// TIA Portal project "Onlab" (V16)

(* hardware
DEVICE "S71500/ET200MP station_1"  S7-1500 station
   slot 0: "Rail_0"  Rack  6ES7 590-1***0-0AA0
   slot 1: "PLC_1"  CPU 1515-2 PN  6ES7 515-2AM00-0AB0  V1.8
      slot 3: "CPU display_1"  6ES7591-1BA00-0AA0
      slot 32768: "PROFINET interface_1"  X1
         slot 32769: "Port_1"  X1 P1
         slot 32770: "Port_2"  X1 P2
      slot 33024: "PROFINET interface_2"  X2
         slot 33025: "Port_1"  X2 P1
*)

// ===== PLC "PLC_1"  CPU 1515-2 PN =====

VAR_GLOBAL   // PLC tag table "Default tag table"
   "Start" AT %I0.0 : Bool;
   "ST10_SMD" AT %I0.1 : Bool;
   "ST10_SED" AT %I0.2 : Bool;
   "ST10_SRD" AT %I0.3 : Bool;
   "ST20_SMD" AT %I0.4 : Bool;
   "ST20_SRD" AT %I0.5 : Bool;
   "ST20_SED" AT %I0.6 : Bool;
   "ST30_SMD" AT %I0.7 : Bool;
   "ST30_SRD" AT %I1.0 : Bool;
   "ST30_SED" AT %I1.1 : Bool;
   "Start2" AT %I1.2 : Bool;
END_VAR

DATA_BLOCK "PLC_PRG_DB"   // DB1
{ S7_Optimized_Access := 'TRUE' }
VERSION : 0.1
   VAR
      startp : Bool;
      start2p : Bool;
      st10smdp : Bool;
      st10srdp : Bool;
      st10sedp : Bool;
      st20smdp : Bool;
      st20srdp : Bool;
      st20sedp : Bool;
      st30smdp : Bool;
      st30srdp : Bool;
      st30sedp : Bool;
      st40smdp : Bool;
      st40srdp : Bool;
      st40sedp : Bool;
      st20recrdy : Bool;
      st30recrdy : Bool;
      st40recrdy : Bool;
   END_VAR
BEGIN
END_DATA_BLOCK

DATA_BLOCK "ST10"   // DB9
{ S7_Optimized_Access := 'TRUE' }
VERSION : 0.1
// stored: InstanceOfName CB
"CB"
BEGIN
END_DATA_BLOCK

DATA_BLOCK "ST20"   // DB10
{ S7_Optimized_Access := 'TRUE' }
VERSION : 0.1
// stored: InstanceOfName CB
"CB"
BEGIN
END_DATA_BLOCK

DATA_BLOCK "ST30"   // DB11
{ S7_Optimized_Access := 'TRUE' }
VERSION : 0.1
// stored: InstanceOfName CB
"CB"
BEGIN
END_DATA_BLOCK

DATA_BLOCK "ST40_db"   // DB12
{ S7_Optimized_Access := 'TRUE' }
VERSION : 0.1
// stored: InstanceOfName CB
"CB"
BEGIN
END_DATA_BLOCK

DATA_BLOCK "ST50"   // DB13
{ S7_Optimized_Access := 'TRUE' }
VERSION : 0.1
// stored: InstanceOfName CB
"CB"
BEGIN
END_DATA_BLOCK

DATA_BLOCK "ST60"   // DB14
{ S7_Optimized_Access := 'TRUE' }
VERSION : 0.1
// stored: InstanceOfName CB
"CB"
BEGIN
END_DATA_BLOCK

DATA_BLOCK "ST70"   // DB15
{ S7_Optimized_Access := 'TRUE' }
VERSION : 0.1
// stored: InstanceOfName CB
"CB"
BEGIN
END_DATA_BLOCK

// folder: DBk

DATA_BLOCK "ST10_DBaaa"   // DB2
{ S7_Optimized_Access := 'TRUE' }
VERSION : 0.1
   VAR
      Szenzor1 : Bool;   // Optikai szenzor új darab érz. (bemenet)
      Szenzor2 : Bool;   // Lassító szenzor (bemenet)
      Szenzor3 : Bool;   // Megállító szenzor (bemenet)
      NyG : Bool;   // Nyomógomb a pálya elindításához (bemenet)
      Fényv : Bool;   // Fény visszajelzés az operátornak (kimenet)
      Motor100 : Bool;   // Motor 100% sebességgel (kimenet)
      Motor50 : Bool;   // Motor 50% sebességgel (kimenet)
      MotorStop : Bool;   // Motor áll (kimenet)
      NyGPOSEDGE : Bool;   // NyG felfutóél boolja (belső változó)
      Rdy : Bool;   // ST10 Kész új darab fogadására (kimenet)
      Vonalkód : Struct   // Termelésirányításnak átadott adat (kimenet)
         kód : Array[0..7] of Char;
         feldolgozva : Bool;
      END_STRUCT;
      "Kapott adat" : Struct   // Termelésirányítástól kapott információk (bemenet)
         kód : Array[0..7] of Char;
         "új darab" : Bool;
         Levegő : Bool;
         Fény : Bool;
         Visszajáratott : Bool;
      END_STRUCT;
      Állapotok : Array[0..4] of Bool;   // Az állomás állapotai (belső változó)
   END_VAR
BEGIN
   // Állapotok[0] : Várás
   // Állapotok[1] : Motor100
   // Állapotok[2] : Motor50
   // Állapotok[3] : MotorStop
   // Állapotok[4] : Kiadás
END_DATA_BLOCK

DATA_BLOCK "ST20_DBaaa"   // DB3
{ S7_Optimized_Access := 'TRUE' }
VERSION : 0.1
   VAR
      Szenzor1 : Bool := false;   // Lassító szenzor (bemenet)
      Szenzor2 : Bool := false;   // Megállító szenzor (bemenet)
      Vízsz : Bool := false;   // Végállás érz. (bemenet)
      Függ : Bool := false;   // Végállás érz. (bemenet)
      Motor100 : Bool := false;   // Motor 100% sebességgel (kimenet)
      Motor50 : Bool := false;   // Motor 50% sebességgel (kimenet)
      MotorStop : Bool := false;   // Motor áll (kimenet)
      NyGPOSEDGE : Bool := false;   // NyG felfutóél boolja (belső változó)
      Rdy : Bool;   // ST20 Kész új darab fogadására (kimenet)
      Vonalkód : Struct   // Termelésirányításnak átadott adat (kimenet)
         kód : Array[0..7] of Char;
         feldolgozva : Bool;
      END_STRUCT;
      "Kapott adat" : Struct   // Termelésirányítástól kapott információk (bemenet)
         kód : Array[0..7] of Char;
         "új darab" : Bool;
         Levegő : Bool;
         Fény : Bool;
         Visszajáratott : Bool;
      END_STRUCT;
      Állapotok : Array[0..5] of Bool;   // Az állomás állapotai (belső változó)
   END_VAR
BEGIN
   // Állapotok[0] : Várás
   // Állapotok[1] : Motor100
   // Állapotok[2] : Motor50
   // Állapotok[3] : MotorStop
   // Állapotok[4] : ST30 felé
   // Állapotok[5] : ST60 felé
END_DATA_BLOCK

DATA_BLOCK "ST30_DBaaa"   // DB4
{ S7_Optimized_Access := 'TRUE' }
VERSION : 0.1
   VAR
      Szenzor1 : Bool := false;   // Lassító szenzor (bemenet)
      Szenzor2 : Bool := false;   // Megállító szenzor (bemenet)
      Vízsz : Bool := false;   // Végállás érz. (bemenet)
      Függ : Bool := false;   // Végállás érz. (bemenet)
      Motor100 : Bool := false;   // Motor 100% sebességgel (kimenet)
      Motor50 : Bool := false;   // Motor 50% sebességgel (kimenet)
      MotorStop : Bool := false;   // Motor áll (kimenet)
      NyGPOSEDGE : Bool := false;   // NyG felfutóél boolja (belső változó)
      Rdy : Bool;   // ST30 Kész új darab fogadására (kimenet)
      Vonalkód : Struct   // Termelésirányításnak átadott adat (kimenet)
         kód : Array[0..7] of Char;
         feldolgozva : Bool;
      END_STRUCT;
      "Kapott adat" : Struct   // Termelésirányítástól kapott információk (bemenet)
         kód : Array[0..7] of Char;
         "új darab" : Bool;
         Levegő : Bool;
         Fény : Bool;
         Visszajáratott : Bool;
      END_STRUCT;
      Állapotok : Array[0..5] of Bool;   // Az állomás állapotai (belső változó)
   END_VAR
BEGIN
   // Állapotok[0] : Várás
   // Állapotok[1] : Motor100
   // Állapotok[2] : Motor50
   // Állapotok[3] : MotorStop
   // Állapotok[4] : ST30 felé
   // Állapotok[5] : ST60 felé
END_DATA_BLOCK

DATA_BLOCK "ST40_DBaaa"   // DB5
{ S7_Optimized_Access := 'TRUE' }
VERSION : 0.1
   VAR
      Szenzor1 : Bool := false;   // Lassító szenzor (bemenet)
      Szenzor2 : Bool := false;   // Megállító szenzor (bemenet)
      Felső : Bool := false;   // Végállás érz. (bemenet)
      Alsó : Bool := false;   // Végállás érz. (bemenet)
      Motor100 : Bool := false;   // Motor 100% sebességgel (kimenet)
      Motor50 : Bool := false;   // Motor 50% sebességgel (kimenet)
      MotorStop : Bool := false;   // Motor áll (kimenet)
      NyGPOSEDGE : Bool := false;   // NyG felfutóél boolja (belső változó)
      Rdy : Bool;   // ST40 Kész új darab fogadására (kimenet)
      KiadásRdy : Bool;
      Vonalkód : Struct   // Termelésirányításnak átadott adat (kimenet)
         kód : Array[0..7] of Char;
         feldolgozva : Bool;
      END_STRUCT;
      "Kapott adat" : Struct   // Termelésirányítástól kapott információk (bemenet)
         kód : Array[0..7] of Char;
         "új darab" : Bool;
         Levegő : Bool;
         Fény : Bool;
         Visszajáratott : Bool;
      END_STRUCT;
      Állapotok : Array[0..5] of Bool;   // Az állomás állapotai (belső változó)
   END_VAR
BEGIN
   // Állapotok[0] : Várás (Az állomás fent van ST30-nál)
   // Állapotok[1] : Motor100
   // Állapotok[2] : Motor50
   // Állapotok[3] : MotorStop
   // Állapotok[4] : ST30 felé
   // Állapotok[5] : ST60 felé
END_DATA_BLOCK

DATA_BLOCK "ST50_DBaaa"   // DB6
{ S7_Optimized_Access := 'TRUE' }
VERSION : 0.1
   VAR
      Szenzor1 : Bool;   // Optikai szenzor új darab érz. (bemenet)
      Szenzor2 : Bool;   // Lassító szenzor (bemenet)
      Motor100 : Bool;   // Motor 100% sebességgel (kimenet)
      Motor50 : Bool;   // Motor 50% sebességgel (kimenet)
      MotorStop : Bool;   // Motor áll (kimenet)
      NyGPOSEDGE : Bool;   // NyG felfutóél boolja (belső változó)
      Rdy : Bool;   // ST10 Kész új darab fogadására (kimenet)
      Vonalkód : Struct   // Termelésirányításnak átadott adat (kimenet)
         kód : Array[0..7] of Char;
         feldolgozva : Bool;
      END_STRUCT;
      "Kapott adat" : Struct   // Termelésirányítástól kapott információk (bemenet)
         kód : Array[0..7] of Char;
         "új darab" : Bool;
         Levegő : Bool;
         Fény : Bool;
         Visszajáratott : Bool;
      END_STRUCT;
      Állapotok : Array[0..4] of Bool;   // Az állomás állapotai (belső változó)
   END_VAR
BEGIN
   // Állapotok[0] : Várás
   // Állapotok[1] : Motor100
   // Állapotok[2] : Motor50
   // Állapotok[3] : MotorStop
   // Állapotok[4] : Kiadás
END_DATA_BLOCK

DATA_BLOCK "ST60_DBaaa"   // DB7
{ S7_Optimized_Access := 'TRUE' }
VERSION : 0.1
   VAR
      Szenzor1 : Bool;   // Optikai szenzor új darab érz. (bemenet)
      Szenzor2 : Bool;   // Lassító szenzor (bemenet)
      Motor100 : Bool;   // Motor 100% sebességgel (kimenet)
      Motor50 : Bool;   // Motor 50% sebességgel (kimenet)
      MotorStop : Bool;   // Motor áll (kimenet)
      NyGPOSEDGE : Bool;   // NyG felfutóél boolja (belső változó)
      Rdy : Bool;   // ST10 Kész új darab fogadására (kimenet)
      RagasztásS : Bool;   // RagasztásStart (kimenet)
      RagasztásM : Bool;   // Ragasztás megszakítás (ki kell sorolni a minőségellenőrző állomásra) (kimenet)
      HibásP : Bool;   // Hibás parancs (bemenet)
      "Ragasztás alatt" : Bool;   // (bemenet)
      SikeresR : Bool;   // Sikeres ragasztás (bemenet)
      SikertelenR : Bool;   // Sikertelen ragasztás (bemenet)
      ProgramSz : Int;   // Programszám (Int) „1”:Levegőre kötő ragasztás ; „2”:UV-ra kötő ragasztás (bemenet és kimenet)
      Vonalkód : Struct   // Termelésirányításnak átadott adat (kimenet)
         kód : Array[0..7] of Char;
         feldolgozva : Bool;
      END_STRUCT;
      "Kapott adat" : Struct   // Termelésirányítástól kapott információk (bemenet)
         kód : Array[0..7] of Char;
         "új darab" : Bool;
         Levegő : Bool;
         Fény : Bool;
         Visszajáratott : Bool;
      END_STRUCT;
      Állapotok : Array[0..4] of Bool;   // Az állomás állapotai (belső változó)
   END_VAR
BEGIN
   // Állapotok[0] : Várás
   // Állapotok[1] : Motor100
   // Állapotok[2] : Motor50
   // Állapotok[3] : MotorStop
   // Állapotok[4] : Kiadás
END_DATA_BLOCK

DATA_BLOCK "ST70_DBaaa"   // DB8
{ S7_Optimized_Access := 'TRUE' }
VERSION : 0.1
   VAR
      Szenzor1 : Bool;   // Optikai szenzor új darab érz. (bemenet)
      Szenzor2 : Bool;   // Lassító szenzor (bemenet)
      Motor100 : Bool;   // Motor 100% sebességgel (kimenet)
      Motor50 : Bool;   // Motor 50% sebességgel (kimenet)
      MotorStop : Bool;   // Motor áll (kimenet)
      NyGPOSEDGE : Bool;   // NyG felfutóél boolja (belső változó)
      Rdy : Bool;   // ST10 Kész új darab fogadására (kimenet)
      Nyitás : Bool;   // (ET200-ra kötve) EFAFLEX gyorskapu nyitó (kimenet)
      Zárás : Bool;   // (ET200-ra kötve) EFAFLEX gyorskapu záró (kimenet)
      Nyitva : Bool;   // (ET200-ra kötve) EFAFLEX gyorskapu nyitva van (bemenet)
      Zárva : Bool;   // (ET200-ra kötve) EFAFLEX gyorskapu zárva van (bemenet)
      UVbekapcs : Bool;   // (ET200-ra kötve) UV bekapcsoló (kimenet)
      UVműködik : Bool;   // (ET200-ra kötve) UV működik (bemenet)
      Vonalkód : Struct   // Termelésirányításnak átadott adat (kimenet)
         kód : Array[0..7] of Char;
         feldolgozva : Bool;
      END_STRUCT;
      "Kapott adat" : Struct   // Termelésirányítástól kapott információk (bemenet)
         kód : Array[0..7] of Char;
         "új darab" : Bool;
         Levegő : Bool;
         Fény : Bool;
         Visszajáratott : Bool;
      END_STRUCT;
      Állapotok : Array[0..4] of Bool;   // Az állomás állapotai (belső változó)
   END_VAR
BEGIN
   // Állapotok[0] : Várás
   // Állapotok[1] : Motor100
   // Állapotok[2] : Motor50
   // Állapotok[3] : MotorStop
   // Állapotok[4] : Kiadás
END_DATA_BLOCK

DATA_BLOCK "ACS355_DBaaa"   // DB20
{ S7_Optimized_Access := 'TRUE' }
VERSION : 0.1
   VAR
      Motor100 : Bool;
      Motor30 : Bool;
      MotorStop : Bool;
      MotorDO3 : Bool;
      MotorDO4 : Bool;
   END_VAR
BEGIN
END_DATA_BLOCK

DATA_BLOCK "Láncos pálya_DBaaa"   // DB21
{ S7_Optimized_Access := 'TRUE' }
VERSION : 0.1
   VAR
      Motor100 : Bool;
      Motor50 : Bool;
      MotorStop : Bool;
      MotorDO3 : Bool;
      MotorDO4 : Bool;
   END_VAR
BEGIN
END_DATA_BLOCK

// folder: (top level)

FUNCTION_BLOCK "ST"   // FB1, SCL
{ S7_Optimized_Access := 'TRUE' }
VERSION : 0.1
   VAR_INPUT
      CBSMD : Bool;
      CBSRD : Bool;
      CBSED : Bool;
      CBSend : Bool;
      CBEnable : Bool;
      CBManMotor100 : Bool;
      CBManMotor30 : Bool;
      CBManMotorStop : Bool;
      CBManSendRdy : Bool;
      CBManSending : Bool;
      CBManRecRdy : Bool;
      CBManReceiving : Bool;
      CBManual : Bool;
      TTEnable : Bool;
      TTManual : Bool;
      TTManualMotor100 : Bool;
      TTManualMotor30 : Bool;
      TTManualMotorStop : Bool;
      TTManualMotorDir : Bool;
      TTManualVertState : Bool;
      TTManualHorState : Bool;
      TTHED : Bool;
      TTHRD : Bool;
      TTVED : Bool;
      TTVRD : Bool;
      TTRotVert : Bool;
      TTRotHor : Bool;
      LEnable : Bool;
      LManual : Bool;
      LManualMotor : Bool;
      LManualDir : Bool;
      LManualUpState : Bool;
      LManualDownState : Bool;
      LGoUp : Bool;
      LGoDown : Bool;
      LDED : Bool;
      LUED : Bool;
   END_VAR
   VAR_OUTPUT
      CBMotor100 : Bool;
      CBMotor30 : Bool;
      CBMotorStop : Bool;
      TTMotor100 : Bool;
      TTMotor30 : Bool;
      TTMotorStop : Bool;
      TTMotorDir : Bool;
      TTVertState : Bool;
      TTHorState : Bool;
      LMotor : Bool;
      LDir : Bool;
      LUpState : Bool;
      LDownState : Bool;
   END_VAR
   VAR_IN_OUT
      CBSendRdyVert : Bool;
      CBSendRdyHor : Bool;
      CBPrevSendRdyVert : Bool;
      CBPrevSendRdyHor : Bool;
      CBRecRdyVert : Bool;
      CBRecRdyHor : Bool;
      CBNextRecRdyVert : Bool;
      CBNextRecRdyHor : Bool;
   END_VAR
   VAR
      CB_Instance : "CB";
      TT_Instance : "TT";
      L_Instance : "L";
      CBDirSet : Bool;
      CBHalt : Bool;
      CBSendRdyActual : Bool;
      PrevSendRdyActual : Bool;
      RecRdyActual : Bool;
      NextRecRdyActual : Bool;
   END_VAR
BEGIN
   #TT_Instance(Enable := #TTEnable,
                Manual := #TTManual,
                ManualMotor100 := #TTManualMotor100,
                ManualMotor30 := #TTManualMotor30,
                ManualMotorStop := #TTManualMotorStop,
                ManualMotorDir := #TTManualMotorDir,
                ManualVertState := #TTManualVertState,
                ManualHorState := #TTManualHorState,
                HED := #TTHED,
                HRD := #TTHRD,
                VED := #TTVED,
                VRD := #TTVRD,
                RotVert := #TTRotVert,
                RotHor := #TTRotHor,
                Motor100 => #TTMotor100,
                Motor30 => #TTMotor30,
                MotorStop => #TTMotorStop,
                MotorDir => #TTMotorDir,
                VertState => #TTVertState,
                HorState => #TTHorState);

   #CBDirSet := #TT_Instance.VertState OR #TT_Instance.HorState; //ha a futószalag nem mozog, akkor beállítja a megfelelő irányt, amivel át lehet kapcsolni a CB interfészét a másik CB-khez.
   IF #CBDirSet THEN
       IF #TT_Instance.VertState THEN
           #CBHalt := FALSE; //CB letiltás ne legyen
           #CBSendRdyActual := #CBSendRdyVert; //egyik CB
           #PrevSendRdyActual := #CBPrevSendRdyVert; //egyik CB
           #RecRdyActual := #CBRecRdyVert; //egyik CB
           #NextRecRdyActual := #CBNextRecRdyVert; //egyik CB
       ELSE
           #CBHalt := FALSE; //CB letiltás ne legyen
           #CBSendRdyActual := #CBSendRdyHor; //másik CB
           #PrevSendRdyActual := #CBPrevSendRdyHor; //másik CB
           #RecRdyActual := #CBRecRdyHor; //másik CB
           #NextRecRdyActual := #CBNextRecRdyHor; //másik CB
       END_IF;
   ELSE
       #CBHalt := TRUE; //CB letiltás legyen, amíg a forgatóasztal mozog.
   END_IF;

   #CB_Instance(SMD := #CBSMD,
                SRD := #CBSRD,
                SED := #CBSED,
                Send := #CBSend,
                Enable := #CBEnable AND NOT(#CBHalt),
                ManMotor100 := #CBManMotor100,
                ManMotor30 := #CBManMotor30,
                ManMotorStop := #CBManMotorStop,
                ManSendRdy := #CBManRecRdy,
                ManSending := #CBManSending,
                ManRecRdy := #CBManRecRdy,
                ManReceiving := #CBManReceiving,
                Manual := #CBManual,
                Motor100 => #CBMotor100,
                Motor30 => #CBMotor30,
                MotorStop => #CBMotorStop,
                SendRdy := #CBSendRdyActual,
                PrevSendRdy := #PrevSendRdyActual,
                RecRdy := #RecRdyActual,
                NextRecRdy := #NextRecRdyActual);

   #L_Instance(Enable:=#LEnable,
                Manual:=#LManual,
                ManualMotor:=#LManualMotor,
                ManualDir:=#LManualDir,
                ManualUpState:=#LManualUpState,
                ManualDownState:=#LManualDownState,
                GoUp:=#LGoUp,
                GoDown:=#LGoDown,
                DED:=#LDED,
                UED:=#LUED,
                Motor=>#LMotor,
                Dir=>#LDir,
                UpState=>#LUpState,
                DownState=>#LDownState);
END_FUNCTION_BLOCK

FUNCTION_BLOCK "STB"   // FB1, SCL
{ S7_Optimized_Access := 'TRUE' }
VERSION : 0.1
   VAR_INPUT
      CBSMD : Bool;
      CBSRD : Bool;
      CBSED : Bool;
      CBSend : Bool;
      CBEnable : Bool;
      CBManMotor100 : Bool;
      CBManMotor30 : Bool;
      CBManMotorStop : Bool;
      CBManSendRdy : Bool;
      CBManSending : Bool;
      CBManRecRdy : Bool;
      CBManReceiving : Bool;
      CBManual : Bool;
      TTEnable : Bool;
      TTManual : Bool;
      TTManualMotor100 : Bool;
      TTManualMotor30 : Bool;
      TTManualMotorStop : Bool;
      TTManualMotorDir : Bool;
      TTManualVertState : Bool;
      TTManualHorState : Bool;
      TTHED : Bool;
      TTHRD : Bool;
      TTVED : Bool;
      TTVRD : Bool;
      TTRotVert : Bool;
      TTRotHor : Bool;
      LEnable : Bool;
      LManual : Bool;
      LManualMotor : Bool;
      LManualDir : Bool;
      LManualUpState : Bool;
      LManualDownState : Bool;
      LGoUp : Bool;
      LGoDown : Bool;
      LDED : Bool;
      LUED : Bool;
   END_VAR
   VAR_OUTPUT
      CBMotor100 : Bool;
      CBMotor30 : Bool;
      CBMotorStop : Bool;
      TTMotor100 : Bool;
      TTMotor30 : Bool;
      TTMotorStop : Bool;
      TTMotorDir : Bool;
      TTVertState : Bool;
      TTHorState : Bool;
      LMotor : Bool;
      LDir : Bool;
      LUpState : Bool;
      LDownState : Bool;
   END_VAR
   VAR_IN_OUT
      CBSendRdyVert : Bool;
      CBSendRdyHor : Bool;
      CBPrevSendRdyVert : Bool;
      CBPrevSendRdyHor : Bool;
      CBRecRdyVert : Bool;
      CBRecRdyHor : Bool;
      CBNextRecRdyVert : Bool;
      CBNextRecRdyHor : Bool;
   END_VAR
   VAR
      CB_Instance : "CB";
      TT_Instance : "TT";
      L_Instance : "L";
      CBDirSet : Bool;
      CBHalt : Bool;
      CBSendRdyActual : Bool;
      PrevSendRdyActual : Bool;
      RecRdyActual : Bool;
      NextRecRdyActual : Bool;
   END_VAR
BEGIN
   #TT_Instance(Enable := #TTEnable,
                Manual := #TTManual,
                ManualMotor100 := #TTManualMotor100,
                ManualMotor30 := #TTManualMotor30,
                ManualMotorStop := #TTManualMotorStop,
                ManualMotorDir := #TTManualMotorDir,
                ManualVertState := #TTManualVertState,
                ManualHorState := #TTManualHorState,
                HED := #TTHED,
                HRD := #TTHRD,
                VED := #TTVED,
                VRD := #TTVRD,
                RotVert := #TTRotVert,
                RotHor := #TTRotHor,
                Motor100 => #TTMotor100,
                Motor30 => #TTMotor30,
                MotorStop => #TTMotorStop,
                MotorDir => #TTMotorDir,
                VertState => #TTVertState,
                HorState => #TTHorState);

   #CBDirSet := #TT_Instance.VertState OR #TT_Instance.HorState; //ha a futószalag nem mozog, akkor beállítja a megfelelő irányt, amivel át lehet kapcsolni a CB interfészét a másik CB-khez.
   IF #CBDirSet THEN
       IF #TT_Instance.VertState THEN
           #CBHalt := FALSE; //CB letiltás ne legyen
           #CBSendRdyActual := #CBSendRdyVert; //egyik CB
           #PrevSendRdyActual := #CBPrevSendRdyVert; //egyik CB
           #RecRdyActual := #CBRecRdyVert; //egyik CB
           #NextRecRdyActual := #CBNextRecRdyVert; //egyik CB
       ELSE
           #CBHalt := FALSE; //CB letiltás ne legyen
           #CBSendRdyActual := #CBSendRdyHor; //másik CB
           #PrevSendRdyActual := #CBPrevSendRdyHor; //másik CB
           #RecRdyActual := #CBRecRdyHor; //másik CB
           #NextRecRdyActual := #CBNextRecRdyHor; //másik CB
       END_IF;
   ELSE
       #CBHalt := TRUE; //CB letiltás legyen, amíg a forgatóasztal mozog.
   END_IF;

   #CB_Instance(SMD := #CBSMD,
                SRD := #CBSRD,
                SED := #CBSED,
                Send := #CBSend,
                Enable := #CBEnable AND NOT(#CBHalt),
                ManMotor100 := #CBManMotor100,
                ManMotor30 := #CBManMotor30,
                ManMotorStop := #CBManMotorStop,
                ManSendRdy := #CBManRecRdy,
                ManSending := #CBManSending,
                ManRecRdy := #CBManRecRdy,
                ManReceiving := #CBManReceiving,
                Manual := #CBManual,
                Motor100 => #CBMotor100,
                Motor30 => #CBMotor30,
                MotorStop => #CBMotorStop,
                SendRdy := #CBSendRdyActual,
                PrevSendRdy := #PrevSendRdyActual,
                RecRdy := #RecRdyActual,
                NextRecRdy := #NextRecRdyActual);

   #L_Instance(Enable:=#LEnable,
                Manual:=#LManual,
                ManualMotor:=#LManualMotor,
                ManualDir:=#LManualDir,
                ManualUpState:=#LManualUpState,
                ManualDownState:=#LManualDownState,
                GoUp:=#LGoUp,
                GoDown:=#LGoDown,
                DED:=#LDED,
                UED:=#LUED,
                Motor=>#LMotor,
                Dir=>#LDir,
                UpState=>#LUpState,
                DownState=>#LDownState);
END_FUNCTION_BLOCK

FUNCTION_BLOCK "STG"   // FB1, SCL
{ S7_Optimized_Access := 'TRUE' }
VERSION : 0.1
   VAR_INPUT
      CBSMD : Bool;
      CBSRD : Bool;
      CBSED : Bool;
      CBSend : Bool;
      CBEnable : Bool;
      CBManMotor100 : Bool;
      CBManMotor30 : Bool;
      CBManMotorStop : Bool;
      CBManSendRdy : Bool;
      CBManSending : Bool;
      CBManRecRdy : Bool;
      CBManReceiving : Bool;
      CBManual : Bool;
      TTEnable : Bool;
      TTManual : Bool;
      TTManualMotor100 : Bool;
      TTManualMotor30 : Bool;
      TTManualMotorStop : Bool;
      TTManualMotorDir : Bool;
      TTManualVertState : Bool;
      TTManualHorState : Bool;
      TTHED : Bool;
      TTHRD : Bool;
      TTVED : Bool;
      TTVRD : Bool;
      TTRotVert : Bool;
      TTRotHor : Bool;
      LEnable : Bool;
      LManual : Bool;
      LManualMotor : Bool;
      LManualDir : Bool;
      LManualUpState : Bool;
      LManualDownState : Bool;
      LGoUp : Bool;
      LGoDown : Bool;
      LDED : Bool;
      LUED : Bool;
   END_VAR
   VAR_OUTPUT
      CBMotor100 : Bool;
      CBMotor30 : Bool;
      CBMotorStop : Bool;
      TTMotor100 : Bool;
      TTMotor30 : Bool;
      TTMotorStop : Bool;
      TTMotorDir : Bool;
      TTVertState : Bool;
      TTHorState : Bool;
      LMotor : Bool;
      LDir : Bool;
      LUpState : Bool;
      LDownState : Bool;
   END_VAR
   VAR_IN_OUT
      CBSendRdyVert : Bool;
      CBSendRdyHor : Bool;
      CBPrevSendRdyVert : Bool;
      CBPrevSendRdyHor : Bool;
      CBRecRdyVert : Bool;
      CBRecRdyHor : Bool;
      CBNextRecRdyVert : Bool;
      CBNextRecRdyHor : Bool;
   END_VAR
   VAR
      CB_Instance : "CB";
      TT_Instance : "TT";
      L_Instance : "L";
      CBDirSet : Bool;
      CBHalt : Bool;
      CBSendRdyActual : Bool;
      PrevSendRdyActual : Bool;
      RecRdyActual : Bool;
      NextRecRdyActual : Bool;
   END_VAR
BEGIN
   #TT_Instance(Enable := #TTEnable,
                Manual := #TTManual,
                ManualMotor100 := #TTManualMotor100,
                ManualMotor30 := #TTManualMotor30,
                ManualMotorStop := #TTManualMotorStop,
                ManualMotorDir := #TTManualMotorDir,
                ManualVertState := #TTManualVertState,
                ManualHorState := #TTManualHorState,
                HED := #TTHED,
                HRD := #TTHRD,
                VED := #TTVED,
                VRD := #TTVRD,
                RotVert := #TTRotVert,
                RotHor := #TTRotHor,
                Motor100 => #TTMotor100,
                Motor30 => #TTMotor30,
                MotorStop => #TTMotorStop,
                MotorDir => #TTMotorDir,
                VertState => #TTVertState,
                HorState => #TTHorState);

   #CBDirSet := #TT_Instance.VertState OR #TT_Instance.HorState; //ha a futószalag nem mozog, akkor beállítja a megfelelő irányt, amivel át lehet kapcsolni a CB interfészét a másik CB-khez.
   IF #CBDirSet THEN
       IF #TT_Instance.VertState THEN
           #CBHalt := FALSE; //CB letiltás ne legyen
           #CBSendRdyActual := #CBSendRdyVert; //egyik CB
           #PrevSendRdyActual := #CBPrevSendRdyVert; //egyik CB
           #RecRdyActual := #CBRecRdyVert; //egyik CB
           #NextRecRdyActual := #CBNextRecRdyVert; //egyik CB
       ELSE
           #CBHalt := FALSE; //CB letiltás ne legyen
           #CBSendRdyActual := #CBSendRdyHor; //másik CB
           #PrevSendRdyActual := #CBPrevSendRdyHor; //másik CB
           #RecRdyActual := #CBRecRdyHor; //másik CB
           #NextRecRdyActual := #CBNextRecRdyHor; //másik CB
       END_IF;
   ELSE
       #CBHalt := TRUE; //CB letiltás legyen, amíg a forgatóasztal mozog.
   END_IF;

   #CB_Instance(SMD := #CBSMD,
                SRD := #CBSRD,
                SED := #CBSED,
                Send := #CBSend,
                Enable := #CBEnable AND NOT(#CBHalt),
                ManMotor100 := #CBManMotor100,
                ManMotor30 := #CBManMotor30,
                ManMotorStop := #CBManMotorStop,
                ManSendRdy := #CBManRecRdy,
                ManSending := #CBManSending,
                ManRecRdy := #CBManRecRdy,
                ManReceiving := #CBManReceiving,
                Manual := #CBManual,
                Motor100 => #CBMotor100,
                Motor30 => #CBMotor30,
                MotorStop => #CBMotorStop,
                SendRdy := #CBSendRdyActual,
                PrevSendRdy := #PrevSendRdyActual,
                RecRdy := #RecRdyActual,
                NextRecRdy := #NextRecRdyActual);

   #L_Instance(Enable:=#LEnable,
                Manual:=#LManual,
                ManualMotor:=#LManualMotor,
                ManualDir:=#LManualDir,
                ManualUpState:=#LManualUpState,
                ManualDownState:=#LManualDownState,
                GoUp:=#LGoUp,
                GoDown:=#LGoDown,
                DED:=#LDED,
                UED:=#LUED,
                Motor=>#LMotor,
                Dir=>#LDir,
                UpState=>#LUpState,
                DownState=>#LDownState);
END_FUNCTION_BLOCK

FUNCTION_BLOCK "STY"   // FB1, SCL
{ S7_Optimized_Access := 'TRUE' }
VERSION : 0.1
   VAR_INPUT
      CBSMD : Bool;
      CBSRD : Bool;
      CBSED : Bool;
      CBSend : Bool;
      CBEnable : Bool;
      CBManMotor100 : Bool;
      CBManMotor30 : Bool;
      CBManMotorStop : Bool;
      CBManSendRdy : Bool;
      CBManSending : Bool;
      CBManRecRdy : Bool;
      CBManReceiving : Bool;
      CBManual : Bool;
      TTEnable : Bool;
      TTManual : Bool;
      TTManualMotor100 : Bool;
      TTManualMotor30 : Bool;
      TTManualMotorStop : Bool;
      TTManualMotorDir : Bool;
      TTManualVertState : Bool;
      TTManualHorState : Bool;
      TTHED : Bool;
      TTHRD : Bool;
      TTVED : Bool;
      TTVRD : Bool;
      TTRotVert : Bool;
      TTRotHor : Bool;
      LEnable : Bool;
      LManual : Bool;
      LManualMotor : Bool;
      LManualDir : Bool;
      LManualUpState : Bool;
      LManualDownState : Bool;
      LGoUp : Bool;
      LGoDown : Bool;
      LDED : Bool;
      LUED : Bool;
   END_VAR
   VAR_OUTPUT
      CBMotor100 : Bool;
      CBMotor30 : Bool;
      CBMotorStop : Bool;
      TTMotor100 : Bool;
      TTMotor30 : Bool;
      TTMotorStop : Bool;
      TTMotorDir : Bool;
      TTVertState : Bool;
      TTHorState : Bool;
      LMotor : Bool;
      LDir : Bool;
      LUpState : Bool;
      LDownState : Bool;
   END_VAR
   VAR_IN_OUT
      CBSendRdyVert : Bool;
      CBSendRdyHor : Bool;
      CBPrevSendRdyVert : Bool;
      CBPrevSendRdyHor : Bool;
      CBRecRdyVert : Bool;
      CBRecRdyHor : Bool;
      CBNextRecRdyVert : Bool;
      CBNextRecRdyHor : Bool;
   END_VAR
   VAR
      CB_Instance : "CB";
      TT_Instance : "TT";
      L_Instance : "L";
      CBDirSet : Bool;
      CBHalt : Bool;
      CBSendRdyActual : Bool;
      PrevSendRdyActual : Bool;
      RecRdyActual : Bool;
      NextRecRdyActual : Bool;
   END_VAR
BEGIN
   #TT_Instance(Enable := #TTEnable,
                Manual := #TTManual,
                ManualMotor100 := #TTManualMotor100,
                ManualMotor30 := #TTManualMotor30,
                ManualMotorStop := #TTManualMotorStop,
                ManualMotorDir := #TTManualMotorDir,
                ManualVertState := #TTManualVertState,
                ManualHorState := #TTManualHorState,
                HED := #TTHED,
                HRD := #TTHRD,
                VED := #TTVED,
                VRD := #TTVRD,
                RotVert := #TTRotVert,
                RotHor := #TTRotHor,
                Motor100 => #TTMotor100,
                Motor30 => #TTMotor30,
                MotorStop => #TTMotorStop,
                MotorDir => #TTMotorDir,
                VertState => #TTVertState,
                HorState => #TTHorState);

   #CBDirSet := #TT_Instance.VertState OR #TT_Instance.HorState; //ha a futószalag nem mozog, akkor beállítja a megfelelő irányt, amivel át lehet kapcsolni a CB interfészét a másik CB-khez.
   IF #CBDirSet THEN
       IF #TT_Instance.VertState THEN
           #CBHalt := FALSE; //CB letiltás ne legyen
           #CBSendRdyActual := #CBSendRdyVert; //egyik CB
           #PrevSendRdyActual := #CBPrevSendRdyVert; //egyik CB
           #RecRdyActual := #CBRecRdyVert; //egyik CB
           #NextRecRdyActual := #CBNextRecRdyVert; //egyik CB
       ELSE
           #CBHalt := FALSE; //CB letiltás ne legyen
           #CBSendRdyActual := #CBSendRdyHor; //másik CB
           #PrevSendRdyActual := #CBPrevSendRdyHor; //másik CB
           #RecRdyActual := #CBRecRdyHor; //másik CB
           #NextRecRdyActual := #CBNextRecRdyHor; //másik CB
       END_IF;
   ELSE
       #CBHalt := TRUE; //CB letiltás legyen, amíg a forgatóasztal mozog.
   END_IF;

   #CB_Instance(SMD := #CBSMD,
                SRD := #CBSRD,
                SED := #CBSED,
                Send := #CBSend,
                Enable := #CBEnable AND NOT(#CBHalt),
                ManMotor100 := #CBManMotor100,
                ManMotor30 := #CBManMotor30,
                ManMotorStop := #CBManMotorStop,
                ManSendRdy := #CBManRecRdy,
                ManSending := #CBManSending,
                ManRecRdy := #CBManRecRdy,
                ManReceiving := #CBManReceiving,
                Manual := #CBManual,
                Motor100 => #CBMotor100,
                Motor30 => #CBMotor30,
                MotorStop => #CBMotorStop,
                SendRdy := #CBSendRdyActual,
                PrevSendRdy := #PrevSendRdyActual,
                RecRdy := #RecRdyActual,
                NextRecRdy := #NextRecRdyActual);
END_FUNCTION_BLOCK

FUNCTION_BLOCK "ST40"   // FB1, SCL
{ S7_Optimized_Access := 'TRUE' }
VERSION : 0.1
   VAR_INPUT
      CBSMD : Bool;
      CBSRD : Bool;
      CBSED : Bool;
      CBSend : Bool;
      CBEnable : Bool;
      CBManMotor100 : Bool;
      CBManMotor30 : Bool;
      CBManMotorStop : Bool;
      CBManSendRdy : Bool;
      CBManSending : Bool;
      CBManRecRdy : Bool;
      CBManReceiving : Bool;
      CBManual : Bool;
      TTEnable : Bool;
      TTManual : Bool;
      TTManualMotor100 : Bool;
      TTManualMotor30 : Bool;
      TTManualMotorStop : Bool;
      TTManualMotorDir : Bool;
      TTManualVertState : Bool;
      TTManualHorState : Bool;
      TTHED : Bool;
      TTHRD : Bool;
      TTVED : Bool;
      TTVRD : Bool;
      TTRotVert : Bool;
      TTRotHor : Bool;
      LEnable : Bool;
      LManual : Bool;
      LManualMotor : Bool;
      LManualDir : Bool;
      LManualUpState : Bool;
      LManualDownState : Bool;
      LGoUp : Bool;
      LGoDown : Bool;
      LDED : Bool;
      LUED : Bool;
   END_VAR
   VAR_OUTPUT
      CBMotor100 : Bool;
      CBMotor30 : Bool;
      CBMotorStop : Bool;
      TTMotor100 : Bool;
      TTMotor30 : Bool;
      TTMotorStop : Bool;
      TTMotorDir : Bool;
      TTVertState : Bool;
      TTHorState : Bool;
      LMotor : Bool;
      LDir : Bool;
      LUpState : Bool;
      LDownState : Bool;
   END_VAR
   VAR_IN_OUT
      CBSendRdyVert : Bool;
      CBSendRdyHor : Bool;
      CBPrevSendRdyVert : Bool;
      CBPrevSendRdyHor : Bool;
      CBRecRdyVert : Bool;
      CBRecRdyHor : Bool;
      CBNextRecRdyVert : Bool;
      CBNextRecRdyHor : Bool;
   END_VAR
   VAR
      CB_Instance : "CB";
      TT_Instance : "TT";
      L_Instance : "L";
      CBDirSet : Bool;
      CBHalt : Bool;
      CBSendRdyActual : Bool;
      PrevSendRdyActual : Bool;
      RecRdyActual : Bool;
      NextRecRdyActual : Bool;
   END_VAR
BEGIN
   #TT_Instance(Enable := #TTEnable,
                Manual := #TTManual,
                ManualMotor100 := #TTManualMotor100,
                ManualMotor30 := #TTManualMotor30,
                ManualMotorStop := #TTManualMotorStop,
                ManualMotorDir := #TTManualMotorDir,
                ManualVertState := #TTManualVertState,
                ManualHorState := #TTManualHorState,
                HED := #TTHED,
                HRD := #TTHRD,
                VED := #TTVED,
                VRD := #TTVRD,
                RotVert := #TTRotVert,
                RotHor := #TTRotHor,
                Motor100 => #TTMotor100,
                Motor30 => #TTMotor30,
                MotorStop => #TTMotorStop,
                MotorDir => #TTMotorDir,
                VertState => #TTVertState,
                HorState => #TTHorState);

   #CBDirSet := #TT_Instance.VertState OR #TT_Instance.HorState; //ha a futószalag nem mozog, akkor beállítja a megfelelő irányt, amivel át lehet kapcsolni a CB interfészét a másik CB-khez.
   IF #CBDirSet THEN
       IF #TT_Instance.VertState THEN
           #CBHalt := FALSE; //CB letiltás ne legyen
           #CBSendRdyActual := #CBSendRdyVert; //egyik CB
           #PrevSendRdyActual := #CBPrevSendRdyVert; //egyik CB
           #RecRdyActual := #CBRecRdyVert; //egyik CB
           #NextRecRdyActual := #CBNextRecRdyVert; //egyik CB
       ELSE
           #CBHalt := FALSE; //CB letiltás ne legyen
           #CBSendRdyActual := #CBSendRdyHor; //másik CB
           #PrevSendRdyActual := #CBPrevSendRdyHor; //másik CB
           #RecRdyActual := #CBRecRdyHor; //másik CB
           #NextRecRdyActual := #CBNextRecRdyHor; //másik CB
       END_IF;
   ELSE
       #CBHalt := TRUE; //CB letiltás legyen, amíg a forgatóasztal mozog.
   END_IF;

   #CB_Instance(SMD := #CBSMD,
                SRD := #CBSRD,
                SED := #CBSED,
                Send := #CBSend,
                Enable := #CBEnable AND NOT(#CBHalt),
                ManMotor100 := #CBManMotor100,
                ManMotor30 := #CBManMotor30,
                ManMotorStop := #CBManMotorStop,
                ManSendRdy := #CBManRecRdy,
                ManSending := #CBManSending,
                ManRecRdy := #CBManRecRdy,
                ManReceiving := #CBManReceiving,
                Manual := #CBManual,
                Motor100 => #CBMotor100,
                Motor30 => #CBMotor30,
                MotorStop => #CBMotorStop,
                SendRdy := #CBSendRdyActual,
                PrevSendRdy := #PrevSendRdyActual,
                RecRdy := #RecRdyActual,
                NextRecRdy := #NextRecRdyActual);

   #L_Instance(Enable:=#LEnable,
                Manual:=#LManual,
                ManualMotor:=#LManualMotor,
                ManualDir:=#LManualDir,
                ManualUpState:=#LManualUpState,
                ManualDownState:=#LManualDownState,
                GoUp:=#LGoUp,
                GoDown:=#LGoDown,
                DED:=#LDED,
                UED:=#LUED,
                Motor=>#LMotor,
                Dir=>#LDir,
                UpState=>#LUpState,
                DownState=>#LDownState);
END_FUNCTION_BLOCK

FUNCTION_BLOCK "KP"   // FB2, SCL
{ S7_Optimized_Access := 'TRUE' }
VERSION : 0.1
   VAR_INPUT
      Enable : Bool;
      Manual : Bool;
      ManualOpenState : Bool;
      ManualClosedState : Bool;
      ManualRdy : Bool;
      ManualMotor : Bool;
      ManualDir : Bool;
      Open : Bool;
      Close : Bool;
      OED : Bool;
      CED : Bool;
   END_VAR
   VAR_OUTPUT
      OpenState : Bool;
      ClosedState : Bool;
      Rdy : Bool;
      Motor : Bool;
      Dir : Bool;
   END_VAR
   VAR
      eState : USInt;
   END_VAR
BEGIN
   IF #Enable THEN
       IF NOT (#Manual) THEN
           CASE #eState OF
               0:
                   IF #Open THEN
                       #eState := 1;
                   END_IF;
               1:
                   IF #OED THEN
                       #eState := 2;
                   ELSIF #Close THEN
                       #eState := 3;
                   END_IF;
               2:
                   IF #Close THEN
                       #eState := 3;
                   END_IF;
               3:
                   IF #CED THEN
                       #eState := 0;
                   ELSIF #Open THEN
                       #eState := 1;
                   END_IF;
           END_CASE;

           #Motor := #eState = 1 OR #eState = 3;
           #Dir := #eState = 1;
           #OpenState := #eState = 2;
           #ClosedState := #eState = 0;
           #Rdy := #eState = 0;
       ELSE
           #Motor := #ManualMotor;
           #Dir := #ManualDir;
           #OpenState := #ManualOpenState;
           #ClosedState := #ManualClosedState;
           #Rdy := #ManualRdy;
       END_IF;
   END_IF;
END_FUNCTION_BLOCK

FUNCTION_BLOCK "CB"   // FB4, SCL
{ S7_Optimized_Access := 'TRUE' }
VERSION : 0.1
   VAR_INPUT
      SMD : Bool;
      SRD : Bool;
      SED : Bool;
      Send : Bool;
      Enable : Bool;
      ManMotor100 : Bool;
      ManMotor30 : Bool;
      ManMotorStop : Bool;
      ManSendRdy : Bool;
      ManSending : Bool;
      ManRecRdy : Bool;
      ManReceiving : Bool;
      Manual : Bool;
   END_VAR
   VAR_OUTPUT
      Motor100 : Bool;
      Motor30 : Bool;
      MotorStop : Bool;
   END_VAR
   VAR_IN_OUT
      SendRdy : Bool;
      PrevSendRdy : Bool;
      RecRdy : Bool;
      NextRecRdy : Bool;
   END_VAR
   VAR
      eState : USInt;
      SED_prev : Bool;
   END_VAR
BEGIN
   IF #Enable THEN
       IF NOT(#Manual) THEN
           CASE #eState OF
               0:
                   IF #Send AND (#SMD OR #SRD OR #SED) THEN //Empty State
                       #eState := 1;
                   ELSIF #PrevSendRdy AND NOT(#SMD) AND NOT(#SRD) AND NOT(#SED) THEN
                       #eState := 4;
                   END_IF;
               1:
                   #eState := 2; //köv. blokknak idő reagálásra, hogy a recrdyje be tudjon állni 1-be
               2:
                   IF #NextRecRdy THEN
                       #eState := 3;
                   ELSE
                       #eState := 0;
                   END_IF;
               3:
                   IF #SED_prev AND NOT (#SED) THEN //GoThru state (Motor100)
                       #eState := 0;
                   END_IF;
               4:
                   IF #SRD THEN
                       #eState := 5;
                   END_IF;
               5:
                   IF #SED THEN
                       #eState := 0;
                   END_IF;
               END_CASE;

           #SED_prev := #SED;

           #Motor100 := #eState = 3 OR #eState = 4;
           #Motor30 := #eState = 5;
           #MotorStop := #eState = 0 OR #eState = 1 OR #eState = 2;
           #SendRdy := #eState = 1 OR #eState = 2;
           #RecRdy := #eState = 0 OR #eState = 4;
       ELSE
           #Motor100 := #ManMotor100;
           #Motor30 := #ManMotor30;
           #MotorStop := #ManMotorStop;
           #SendRdy := #ManSendRdy;
           #PrevSendRdy := #ManSending;
           #RecRdy := #ManRecRdy;
           #NextRecRdy := #ManReceiving;
       END_IF;
   ELSE
       #Motor100 := FALSE;
       #Motor30 := FALSE;
       #MotorStop := FALSE;
       #SendRdy := FALSE;
       #PrevSendRdy := FALSE;
       #RecRdy := FALSE;
       #NextRecRdy := FALSE;
   END_IF;
END_FUNCTION_BLOCK

FUNCTION_BLOCK "GLUE"   // FB5, SCL
{ S7_Optimized_Access := 'TRUE' }
VERSION : 0.1
   VAR_IN_OUT
      GlueingSuccess : Bool;
      GlueingFail : Bool;
      Glueing : Bool;
   END_VAR
BEGIN
END_FUNCTION_BLOCK

FUNCTION_BLOCK "TT"   // FB8, SCL
{ S7_Optimized_Access := 'TRUE' }
VERSION : 0.1
   VAR_INPUT
      Enable : Bool;
      Manual : Bool;
      ManualMotor100 : Bool;
      ManualMotor30 : Bool;
      ManualMotorStop : Bool;
      ManualMotorDir : Bool;
      ManualVertState : Bool;
      ManualHorState : Bool;
      HED : Bool;
      HRD : Bool;
      VED : Bool;
      VRD : Bool;
      RotVert : Bool;
      RotHor : Bool;
   END_VAR
   VAR_OUTPUT
      Motor100 : Bool;
      Motor30 : Bool;
      MotorStop : Bool;
      MotorDir : Bool;
      VertState : Bool;
      HorState : Bool;
   END_VAR
   VAR
      eState : USInt;
   END_VAR
BEGIN
   IF #Enable THEN
       IF NOT (#Manual) THEN
           CASE #eState OF
               0:
                   IF #RotVert THEN  //Horizontal state
                       #eState := 1;
                   END_IF;
               1:
                   IF #VRD THEN  // Statement section case 2 to 4
                       #eState := 2;
                   ELSIF #RotHor THEN
                       #eState := 6;
                   END_IF;
               2:
                   IF #VED THEN
                       #eState := 3;
                   ELSIF #RotHor THEN
                       #eState := 6;
                   END_IF;
               3:
                   IF #RotHor THEN
                       #eState := 4;
                   END_IF;
               4:
                   IF #HRD THEN
                       #eState := 5;
                   ELSIF #RotVert THEN
                       #eState := 6;
                   END_IF;
               5:
                   IF #HED THEN
                       #eState := 0;
                   ELSIF #RotVert THEN
                       #eState := 6;
                   END_IF;
               6:
                   IF #RotVert AND NOT (#VRD) THEN
                       #eState := 1;
                   ELSIF #RotVert THEN
                       #eState := 2;
                   ELSIF #RotHor AND NOT (#HRD) THEN
                       #eState := 4;
                   ELSIF #RotHor THEN
                       #eState := 5;
                   END_IF;
           END_CASE;

           #Motor100 := #eState = 1 OR #eState = 4;
           #Motor30 := #eState = 2 OR #eState = 5;
           #MotorStop := #eState = 0 OR #eState = 3;
           #MotorDir := #eState = 0 OR #eState = 1 OR #eState = 2;
           #VertState := #eState = 3;
           #HorState := #eState = 0;
       ELSE
           #Motor100 := #ManualMotor100;
           #Motor30 := #ManualMotor30;
           #MotorStop := #ManualMotorStop;
           #MotorDir := #ManualMotorDir;
           #VertState := #ManualVertState;
           #HorState := #ManualHorState;
       END_IF;
   END_IF;
END_FUNCTION_BLOCK

FUNCTION_BLOCK "CT"   // FB9, SCL
{ S7_Optimized_Access := 'TRUE' }
VERSION : 0.1
   VAR_INPUT
      Enable : Bool;
      Manual : Bool;
      ManualMotor : Bool;
      ManualDir : Bool;
      ManualEndState : Bool;
      ManualStartState : Bool;
      GotoEnd : Bool;
      GotoStart : Bool;
      SED : Bool;
      EED : Bool;
   END_VAR
   VAR_OUTPUT
      Motor : Bool;
      Dir : Bool;
      EndState : Bool;
      StartState : Bool;
   END_VAR
   VAR
      eState : USInt;
   END_VAR
BEGIN
   IF #Enable THEN
       IF NOT (#Manual) THEN
           CASE #eState OF
               0:
                   IF #GotoEnd THEN
                       #eState := 1;
                   END_IF;
               1:
                   IF #EED THEN
                       #eState := 2;
                   ELSIF #GotoStart THEN
                       #eState := 3;
                   END_IF;
               2:
                   IF #GotoStart THEN
                       #eState := 3;
                   END_IF;
               3:
                   IF #SED THEN
                       #eState := 0;
                   ELSIF #GotoEnd THEN
                       #eState := 1;
                   END_IF;
           END_CASE;

           #Motor := #eState = 1 OR #eState = 3;
           #Dir := #eState = 1;
           #StartState := #eState = 0;
           #EndState := #eState = 2;
       ELSE
           #Motor := #ManualMotor;
           #Dir := #ManualDir;
           #StartState := #ManualStartState;
           #EndState := #ManualEndState;
       END_IF;
   END_IF;
END_FUNCTION_BLOCK

FUNCTION_BLOCK "L"   // FB10, SCL
{ S7_Optimized_Access := 'TRUE' }
VERSION : 0.1
   VAR_INPUT
      Enable : Bool;
      Manual : Bool;
      ManualMotor : Bool;
      ManualDir : Bool;
      ManualUpState : Bool;
      ManualDownState : Bool;
      GoUp : Bool;
      GoDown : Bool;
      DED : Bool;
      UED : Bool;
   END_VAR
   VAR_OUTPUT
      Motor : Bool;
      Dir : Bool;
      UpState : Bool;
      DownState : Bool;
   END_VAR
   VAR
      eState : USInt;
   END_VAR
BEGIN
   IF #Enable THEN
       IF NOT (#Manual) THEN
           CASE #eState OF
               0:
                   IF #GoUp THEN
                       #eState := 1;
                   END_IF;
               1:
                   IF #UED THEN
                       #eState := 2;
                   ELSIF #GoDown THEN
                       #eState := 3;
                   END_IF;
               2:
                   IF #GoDown THEN
                       #eState := 3;
                   END_IF;
               3:
                   IF #DED THEN
                       #eState := 0;
                   ELSIF #GoUp THEN
                       #eState := 1;
                   END_IF;
           END_CASE;

           #Motor := #eState = 1 OR #eState = 3;
           #Dir := #eState = 1;
           #DownState := #eState = 0;
           #UpState := #eState = 2;
       ELSE
           #Motor := #ManualMotor;
           #Dir := #ManualDir;
           #DownState := #ManualUpState;
           #UpState := #ManualDownState;
       END_IF;
   END_IF;
END_FUNCTION_BLOCK

FUNCTION "ACS355" : Void   // FC1, LAD
{ S7_Optimized_Access := 'TRUE' }
VERSION : 0.1
BEGIN

REGION Network 1
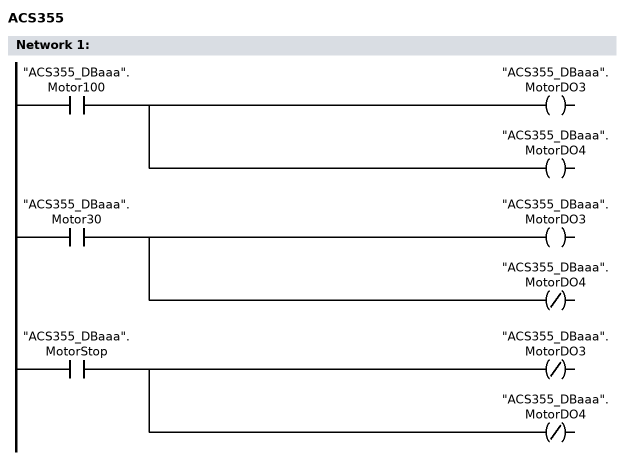
   RUNG wire#powerrail
      Contact( "ACS355_DBaaa".Motor100 )
      wire#w1
      Coil( "ACS355_DBaaa".MotorDO3 )
   END_RUNG
   RUNG wire#w1
      Coil( "ACS355_DBaaa".MotorDO4 )
   END_RUNG
   RUNG wire#powerrail
      Contact( "ACS355_DBaaa".Motor30 )
      wire#w2
      Coil( "ACS355_DBaaa".MotorDO3 )
   END_RUNG
   RUNG wire#w2
      I_Coil( "ACS355_DBaaa".MotorDO4 )
   END_RUNG
   RUNG wire#powerrail
      Contact( "ACS355_DBaaa".MotorStop )
      wire#w3
      I_Coil( "ACS355_DBaaa".MotorDO3 )
   END_RUNG
   RUNG wire#w3
      I_Coil( "ACS355_DBaaa".MotorDO4 )
   END_RUNG
   // the same network as SCL:
   "ACS355_DBaaa".MotorDO3 := "ACS355_DBaaa".Motor100;
   "ACS355_DBaaa".MotorDO4 := "ACS355_DBaaa".Motor100;
   "ACS355_DBaaa".MotorDO3 := "ACS355_DBaaa".Motor30;
   "ACS355_DBaaa".MotorDO4 := NOT "ACS355_DBaaa".Motor30;
   "ACS355_DBaaa".MotorDO3 := NOT "ACS355_DBaaa".MotorStop;
   "ACS355_DBaaa".MotorDO4 := NOT "ACS355_DBaaa".MotorStop;
END_REGION
END_FUNCTION

ORGANIZATION_BLOCK "PLC_PRG"   // OB1, SCL, ProgramCycle
TITLE = "Main Program Sweep (Cycle)"
{ S7_Optimized_Access := 'TRUE' }
VERSION : 0.1
   VAR_INPUT
      Initial_Call : Bool;   // Initial call of this OB
      Remanence : Bool;   // =True, if remanent data are available
   END_VAR
BEGIN
   "Start":="PLC_PRG_DB".startp;
   "Start2":="PLC_PRG_DB".start2p;

   "ST10"(Send := "Start",
          Enable := TRUE,
          SMD := "PLC_PRG_DB".st10smdp,
          SRD := "PLC_PRG_DB".st10srdp,
          SED := "PLC_PRG_DB".st10sedp,
          NextRecRdy := "ST20".RecRdy);
   "ST20"(Send := "Start2",
          Enable := TRUE,
          SMD := "PLC_PRG_DB".st20smdp,
          SRD := "PLC_PRG_DB".st20srdp,
          SED := "PLC_PRG_DB".st20sedp,
          NextRecRdy := "ST30".RecRdy,
          SendRdy := "ST30".PrevSendRdy,
          PrevSendRdy := "ST10".SendRdy);
   "ST30"(Enable := TRUE,
          SMD := "PLC_PRG_DB".st30smdp,
          SRD := "PLC_PRG_DB".st30srdp,
          SED := "PLC_PRG_DB".st30sedp,
          NextRecRdy := "ST40".RecRdy,
          SendRdy := "ST40".PrevSendRdy,
          PrevSendRdy := "ST20".SendRdy);
   "ST40"();
END_ORGANIZATION_BLOCK